Xinje XCPPro project, PLC1: XC1-24 (software 3.3j)

PROGRAM Ladder

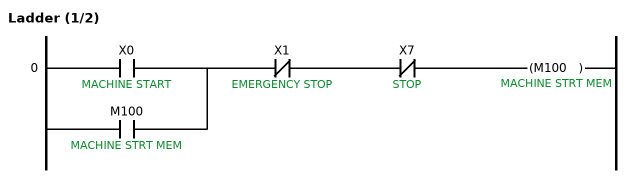
LD     X0	; MACHINE START
OR     M100	; MACHINE STRT MEM
ANI    X1	; EMERGENCY STOP
ANI    X7	; STOP
OUT    M100	; MACHINE STRT MEM

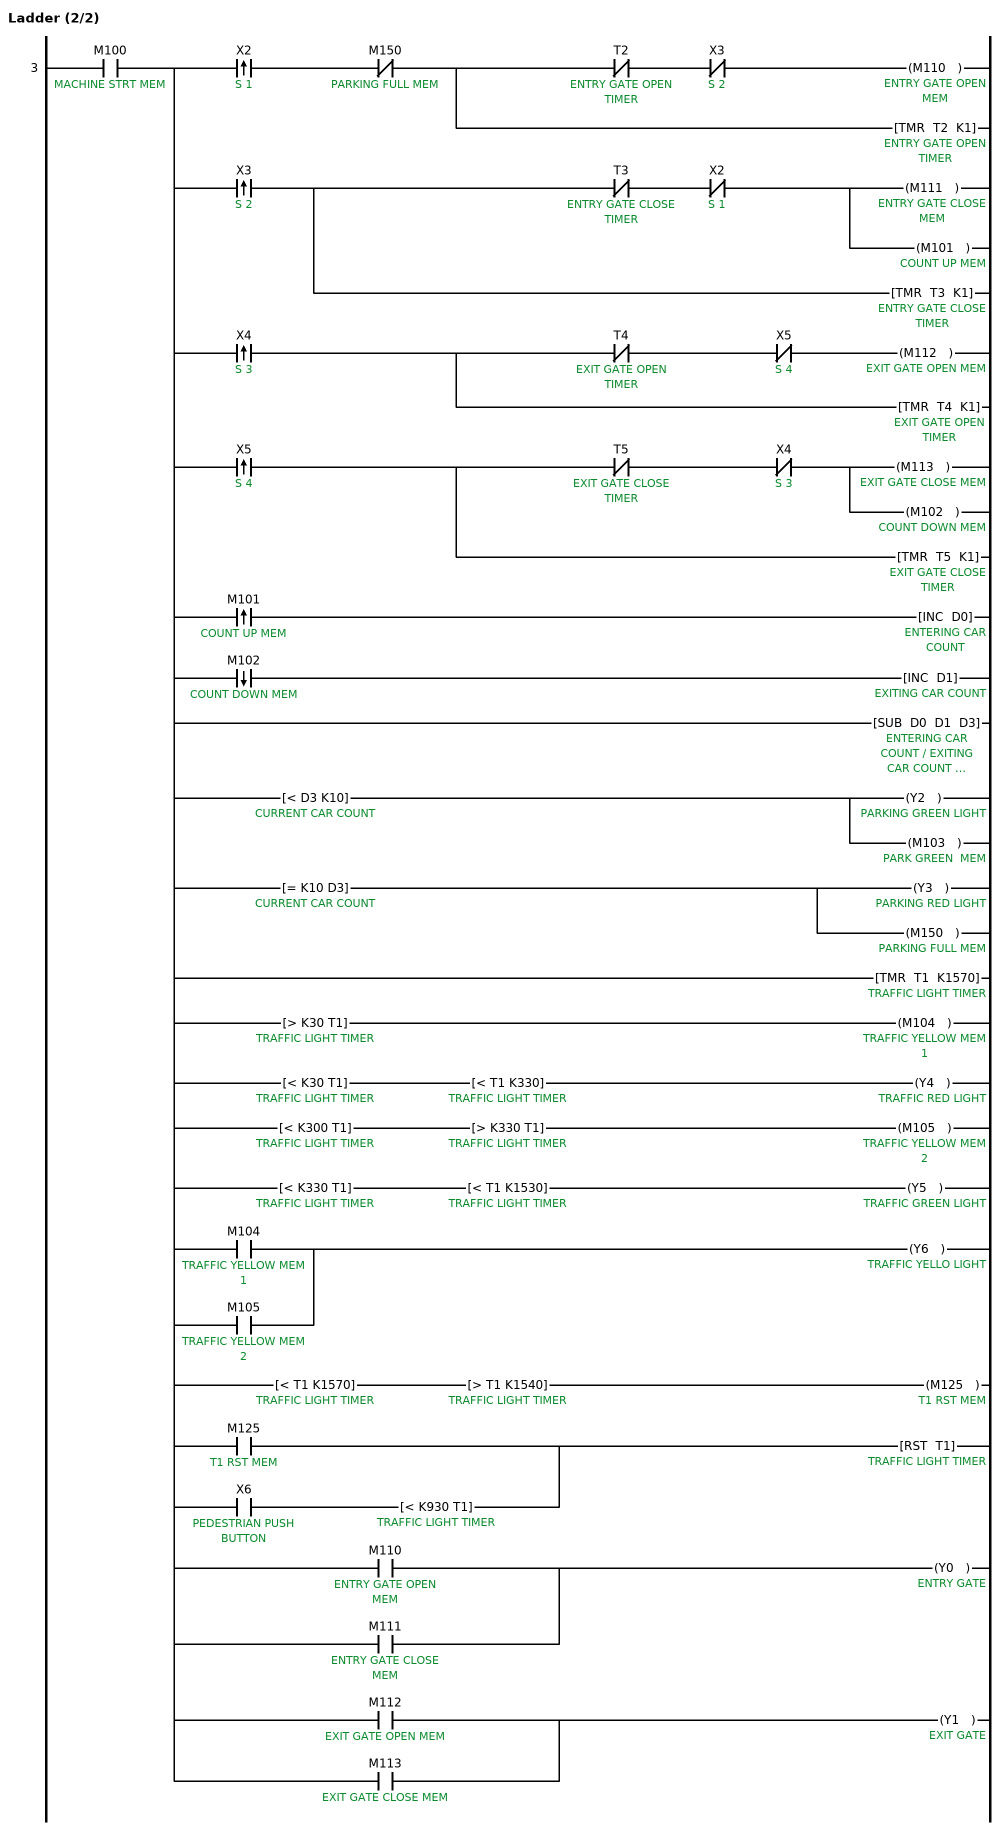
LD     M100	; MACHINE STRT MEM
MPS
ANDP   X2	; S 1
ANI    M150	; PARKING FULL MEM
MPS
ANI    T2	; ENTRY GATE OPEN TIMER
ANI    X3	; S 2
OUT    M110	; ENTRY GATE OPEN MEM
MPP
TMR    T2 K1	; ENTRY GATE OPEN TIMER
MRD
ANDP   X3	; S 2
MPS
ANI    T3	; ENTRY GATE CLOSE TIMER
ANI    X2	; S 1
OUT    M111	; ENTRY GATE CLOSE MEM
OUT    M101	; COUNT UP MEM
MPP
TMR    T3 K1	; ENTRY GATE CLOSE TIMER
MRD
ANDP   X4	; S 3
MPS
ANI    T4	; EXIT GATE OPEN TIMER
ANI    X5	; S 4
OUT    M112	; EXIT GATE OPEN MEM
MPP
TMR    T4 K1	; EXIT GATE OPEN TIMER
MRD
ANDP   X5	; S 4
MPS
ANI    T5	; EXIT GATE CLOSE TIMER
ANI    X4	; S 3
OUT    M113	; EXIT GATE CLOSE MEM
OUT    M102	; COUNT DOWN MEM
MPP
TMR    T5 K1	; EXIT GATE CLOSE TIMER
MRD
ANDP   M101	; COUNT UP MEM
INC    D0	; ENTERING CAR COUNT
MRD
ANDF   M102	; COUNT DOWN MEM
INC    D1	; EXITING CAR COUNT
MRD
SUB    D0 D1 D3	; ENTERING CAR COUNT / EXITING CAR COUNT / CURRENT CAR COUNT
AND<   D3 K10	; CURRENT CAR COUNT
OUT    Y2	; PARKING GREEN LIGHT
OUT    M103	; PARK GREEN  MEM
MRD
AND=   K10 D3	; CURRENT CAR COUNT
OUT    Y3	; PARKING RED LIGHT
OUT    M150	; PARKING FULL MEM
MRD
TMR    T1 K1570	; TRAFFIC LIGHT TIMER
AND>   K30 T1	; TRAFFIC LIGHT TIMER
OUT    M104	; TRAFFIC YELLOW MEM 1
MRD
AND<   K30 T1	; TRAFFIC LIGHT TIMER
AND<   T1 K330	; TRAFFIC LIGHT TIMER
OUT    Y4	; TRAFFIC RED LIGHT
MRD
AND<   K300 T1	; TRAFFIC LIGHT TIMER
AND>   K330 T1	; TRAFFIC LIGHT TIMER
OUT    M105	; TRAFFIC YELLOW MEM 2
MRD
AND<   K330 T1	; TRAFFIC LIGHT TIMER
AND<   T1 K1530	; TRAFFIC LIGHT TIMER
OUT    Y5	; TRAFFIC GREEN LIGHT
MRD
LD     M104	; TRAFFIC YELLOW MEM 1
OR     M105	; TRAFFIC YELLOW MEM 2
ANB
OUT    Y6	; TRAFFIC YELLO LIGHT
MRD
AND<   T1 K1570	; TRAFFIC LIGHT TIMER
AND>   T1 K1540	; TRAFFIC LIGHT TIMER
OUT    M125	; T1 RST MEM
MRD
LD     M125	; T1 RST MEM
LD     X6	; PEDESTRIAN PUSH BUTTON
AND<   K930 T1	; TRAFFIC LIGHT TIMER
ORB
ANB
RST    T1	; TRAFFIC LIGHT TIMER
MRD
LD     M110	; ENTRY GATE OPEN MEM
OR     M111	; ENTRY GATE CLOSE MEM
ANB
OUT    Y0	; ENTRY GATE
MPP
LD     M112	; EXIT GATE OPEN MEM
OR     M113	; EXIT GATE CLOSE MEM
ANB
OUT    Y1	; EXIT GATE

COMMENTS (devices not used above)
Y7	TRAFFIC GREEN LIGHT
Y10	TRAFFIC YELLO LIGHT